PROGRAM MAIN
VAR
	State: E_States;
	i: INT;
	Trigger:ARRAY[1..4]	OF	R_TRIG;
	FB_Sim	:	FB_Sim;
	
	init:BOOL;
END_VAR

IF NOT init THEN
	Floors[1].Mid:=TRUE;
	init:=TRUE;
END_IF

CASE	State	OF
	E_States.Call:
		FOR	i:=1	TO	4	DO
			IF	Floors[i].Call	THEN
				RequestedFloor:=i;
		IF	RequestedFloor>ActualFloor	THEN
			State:=E_States.MoveUp;	
			FB_sim.state:=1;
		ELSIF	RequestedFloor<ActualFloor	THEN
			State:=E_States.MoveDown;	
			FB_sim.state:=16;
		END_IF
			END_IF
		END_FOR
		

	E_States.MoveUp:
		Elevator.MoveUp();
		FOR	i:=1	TO	4	DO
			Trigger[i](clk:=Floors[i].Low);
			IF	Trigger[i].Q	THEN
			//	ActualFloor:=ActualFloor+1;
			END_IF
		END_FOR
		
		IF	ActualFloor=RequestedFloor	THEN
			State:=E_States.SlowDown;
			FB_sim.state:=12;
		END_IF
	E_States.MoveDown:
		Elevator.MoveDown();
		FOR	i:=1	TO	4	DO
			Trigger[i](clk:=Floors[i].High);
			IF	Trigger[i].Q	THEN
			///	ActualFloor:=ActualFloor-1;
			END_IF
		END_FOR
		
		IF	ActualFloor=RequestedFloor	THEN
			State:=E_States.SlowDown;
			FB_sim.state:=27;
		END_IF
		
	E_States.SlowDown:
		Elevator.SlowDown();
		FOR	i:=1	TO	4	DO
			IF	Floors[i].Mid	THEN
				State:=E_States.Stop;
			END_IF
		END_FOR
	E_States.Stop:
		Elevator.Stop();
		State:=E_States.Call;
END_CASE



FB_Sim(Floors:= GVL.Floors, RequestedFloor:= GVL.RequestedFloor, ActualFloor:= GVL.ActualFloor);

END_PROGRAM

(* stored: Version 1.1.0.1, ProductVersion 3.1.4024.9
   POU MAIN: Id {437c88b0-71cb-4e07-9d72-857c04460bf1}, SpecialFunc None *)
